INTERFACE I_Pid

METHOD Reset
END_METHOD

METHOD Update : LREAL
VAR_INPUT
    setpoint    : LREAL;
    measurement : LREAL;
    deltaT      : LREAL;
END_VAR
END_METHOD

END_INTERFACE

(* stored: Version 1.1.0.1
   Itf I_Pid: Id {bce59849-4217-460e-a8ca-3c6683f2e023}
   Method Reset: Id {d4e79a83-5d58-4ac3-9b3f-329dd7730e45}
   Method Update: Id {ebe85e5e-a11d-40e7-b088-27dda55c198b} *)
